{attribute 'qualified_only'}
{attribute 'strict'}
{attribute 'to_string'}
TYPE
ST115_e :
(
    RESET := 0,    // Reset
    INIT := 100,   // Initialisieren 
    READY := 999,  // READY to Start, Init Done 
    START := 1000, // Start Zyklisch
    MOVER_FREE_OP, // Ab here, operation without mover can be done

    // forward to separation, max speed.
	PnP_Hor_ToRotTable,
	
    // down to separation, 1. fast 2. slow (last 20mm)
    // down to separation, 1. fast 2. slow (last 20mm)
	PnP_Ver_RotTableDownFast,
	PnP_Ver_RotTableDownSlow,
	
    // open (pick) --> AS > GS
    // open (pick) --> AS > GS
	PnP_Pick,
	
    // up, 2/3 speed
    // up, 2/3 speed
	PnP_Ver_RotTableUp,
	
    // back to shuttle
	PnP_Hor_ToShuttle,
	
    // separate pice 1 (Check Sensor 110.51)
    // separate pice 2 (Check Sensor 110.51)
	// masked time

    waitOnMover,     // wait until the mover is there
    MOVER_NEEDED_OP, // Since here, a mover in position is needed to perform the action

    // down (with workpiece,) 1. fast 2. slow (press)
    // down (with workpiece,) 1. fast 2. slow (press)
	PnP_Ver_ShuttleDown,
	
    // Check Force during press process
    // Check Force during press process
	PnP_Ver_ShuttleTorque,
	
    // close (releasing) --> GS > AS
    // close (releasing) --> GS > AS
	PnP_Place,
	
    // up, max. speed (3000rpm)
    // up, max. speed (3000rpm)
	PnP_Ver_ShuttleUp,
	
    // Shuttle change

    SYNC_MOVER_LEAVE, // MoverMan need to take the mover
    DONE := 8000,     // Ablauf beendet 
    ERROR := 9000,    // Fehler 
    _max
);
END_TYPE

(* stored: Version 1.1.0.1, ProductVersion 3.1.4024.6
   EnumerationTextList ST115_e: Id {9006f64b-f8ec-4be8-a84e-61da86b4eb29} *)
